TYPE ST_SystemStatus :
	STRUCT
		fPosBuffer   : ARRAY[1..50] OF LREAL; // FIFO position data
		fTenzoBuffer : ARRAY[1..50] OF LREAL; // FIFO tenzo data
		nBufferHead  : INT := 50;             // Index of latest completely written sample
		nSampleCounter    : UDINT := 0;       // Monotonic counter for dropped-sample detection
		nOperationCounter : UDINT := 0;       // Incremented after each completed motion command
		nInterfaceVersion : UDINT := 5;       // MATLAB/PLC ADS contract version
		fTenzoTarOffset   : LREAL := 0.0;     // Calculated tar offset
		fActPosition : LREAL := 0.0;          // Absolute NC axis position
		
		bWorking     : BOOL;                   // PLC occupied; do not send a new test
		bTarWorking  : BOOL;                   // PLC is calculating tare
		bError       : BOOL;                   // Latched application or motion error
		nErrorCode   : UDINT := 0;             // Application error code (0 = no error)
		nAxisErrorID : UDINT := 0;             // Native TwinCAT/NC error ID
		bPowered     : BOOL;                   // Axis power is enabled
		bHoming      : BOOL;                   // Homing command is active
		bHomed       : BOOL;                   // NC axis reports a valid home reference
		bStopped     : BOOL;                   // Axis is at standstill
		bSavedPositionValid : BOOL;            // A return-to-saved reference is available
		nTestPhase   : BYTE := 0;              // 0 idle, 1 pretest, 2 test, 3 post-test
	END_STRUCT
END_TYPE

(* stored: Version 1.1.0.1, ProductVersion 3.1.4024.15
   DUT ST_SystemStatus: Id {1f1ade43-23d7-4c7e-a80f-ab809b514cde} *)
